// TIA Portal V17 export
// export: Created 2022-12-09T10:51:16.9495002Z, ExportSetting WithDefaults, DisplayName Totally Integrated Automation Portal, DisplayVersion V17 Update 5, DisplayName TIA Portal Openness, DisplayVersion V17 Update 5, DisplayName TIA Portal Version Control Interface, DisplayVersion V17, DisplayName Simotion SCOUT TIA, DisplayVersion 5.4.3.0, DisplayName SINAMICS Startdrive Advanced, DisplayVersion V17 SP1, DisplayName SINAMICS Startdrive G130, G150, S120, S150, SINAMICS MV, S210, DisplayVersion V17 SP1, DisplayName SINAMICS Startdrive G110M, G120, G120C, G120D, G120P, G115D, DisplayVersion V17 SP1, DisplayName STEP 7 Professional, DisplayVersion V17 Update 5, DisplayName STEP 7 Safety, DisplayVersion V17, DisplayName WinCC Advanced, DisplayVersion V17 Update 5
TYPE "NDSN_ST_Process"
// stored: IsFailsafeCompliant false
   STRUCT
      i_rw_Temp_arr_ZoneSP : Array[0..17] of Int;
      i_rw_Temp_arr_ZoneActive : Array[0..17] of Int;
      i_rw_Temp_GlobalStandbyDelta : Int;
      i_rw_Temp_ManualStandyDuration : Int;
      i_rw_Temp_AutoEnterStandbyTm : Int;
      i_rw_Temp_AutoHeaterOffTim : Int;
      i_rw_Temp_AutoStandbySourc : Int;
      i_rw_Temp_UnderTempDelta : Int;
      i_rw_Temp_OverTempDelta : Int;
      i_rw_Temp_Unit : Int;
      i_rw_Temp_GlobalSP : Int;
      i_rw_Temp_GlbalHoseSP : Int;
      i_rw_Temp_GlobalGunSP : Int;
      r_rw_Press_SP : Real;
      i_rw_Press_Unit : Int;
      r_rw_Press_MaxPressLimit : Real;
      r_rw_Press_MinPressLimit : Real;
      i_rw_Press_EnableHighLowAlert : Int;
      i_rw_Press_EnableHydrScale : Int;
      r_rw_Press_UnderPressDelta : Real;
      r_rw_Press_OverPressDelta : Real;
      i_rw_Fill_EnableFill : Int;
      i_rw_Fill_TargetFillLevel : Int;
      i_rw_Fill_MaxFillTime : Int;
      i_rw_Fill_AlertStopDelayTime : Int;
      i_rw_Fill_LidOpenAlertTime : Int;
      i_rw_Pump_AutoPump : Int;
      i_rw_Gen_ReadyDelayTime : Int;
      i_rw_Gen_MassUnit : Int;
      i_r_Temp_arr_ZoneActual : Array[0..17] of Int;
      i_r_Temp_arr_ZoneStatus : Array[0..17] of Int;
      r_r_Press_ActualPressure : Real;
      i_r_Press_SensorAlarm : Int;
      i_r_Fill_TankLevel : Int;
      i_r_Gen_SoftwareVersion : Int;
      di_r_Gen_OperationHrs : DInt;
      i_r_Gen_CurrentFaultCode : Int;
      i_r_Gen_arr_SysInventory : Array[0..3] of Int;
      st_r_Device { S7_SetPoint := 'True'} : "NDSN_ST_Inventory";
   END_STRUCT;
END_TYPE
